FUNCTION_BLOCK FB_Schrittbetrieb
VAR_INPUT
	eAblaufStatus:			AblaufStatus;
	eHolStatus:				AblaufStatus;
	eBereitstellStatus:		AblaufStatus;
	bAblaufAktiv:			BOOL;				//Info ob ein Teil bearbetet, geholt oder bereitgestellt werden muss
	
	bAktorPosNIO:			BOOL;				//True wenn ein aktor im handbetrieb verfahren wurde
	
	stStationInfo:			REFERENCE TO ST_Station;
	bRstInPos:				BOOL;
END_VAR
VAR_OUTPUT
	bInQueue:				BOOL;				//Es wurde rueckwaerts in die Queue gefahren und die vorherige Position wurde nicht wieder erreicht
	bAblaufFreigabe:		BOOL;				//Die Aktoren im normalen Ablauf dürfen fahren (Handoverride true) (nur bis Statuswechsel true)
	bSendFalschePosError:	BOOL;				//Aktoren sollen falsche Pos senden
END_VAR
VAR
	aSchrittQueue:			ARRAY[0..Parameter.cGroesseSchrittQueue] OF ST_SchrittQueue;
	nIndex:					INT;
	i:						INT;
	
	nAktPosition:			INT;				//Aktuelle Position in Queue
	nSollAktPos:			INT;				//Welche position andgefahren werden soll (wechselt schon wenn bewegung ausgefuehrt aber Sensoren nicht angeben)
	
	
	ePrevAblaufStatus:		AblaufStatus;
	ePrevHolStatus:			AblaufStatus;	
	ePrevBereitstellStatus:	AblaufStatus;
	
	bBtnSchrittVor:			BOOL;
	bBtnSchrittZurueck:		BOOL;
	
	bSchrittVor:			BOOL;
	bSchrittZurueck:		BOOL;
	bVorBisEnde:			BOOL;
	
	fbSendErrorTrig:		R_TRIG;
END_VAR

//********************************************************************************
//Statuswechsel erkennen
IF			ePrevAblaufStatus <> eAblaufStatus
	OR		ePrevHolStatus <> eHolStatus
	OR		ePrevBereitstellStatus <> eBereitstellStatus THEN
	
	IF			nIndex > 0 THEN
		aSchrittQueue[nIndex-1].bStatuswechsel := TRUE;
	END_IF
	
	bAblaufFreigabe := FALSE;
	
	ePrevAblaufStatus		:= eAblaufStatus;
	ePrevHolStatus			:= eHolStatus;
	ePrevBereitstellStatus	:= eBereitstellStatus;
END_IF

//********************************************************************************
//Handheld
IF			MAIN.fbHandheld.nGewaehlteStation = stStationInfo.nStationsNr THEN
	
	IF			MAIN.bE_Handbetrieb THEN
		
		IF			MAIN.fbHandheld.fbVorTrig.Q THEN
			bBtnSchrittVor := TRUE;
		ELSIF		MAIN.fbHandheld.fbZurueckTrig.Q THEN
			bBtnSchrittZurueck := TRUE;
		END_IF
		
	END_IF
END_IF

//********************************************************************************
//Zurueck zu Start wenn Anlage weiterlaeuft
IF			MAIN.bProduzieren
	AND NOT MAIN.bE_Handbetrieb
	AND		bInQueue
	AND NOT bSchrittZurueck
	AND NOT bSchrittVor THEN
	bVorBisEnde := TRUE;
	bBtnSchrittVor := TRUE;
ELSIF		MAIN.bE_Handbetrieb
	OR	NOT bInQueue THEN
	bVorBisEnde := FALSE;
END_IF

//********************************************************************************
//Aktoren fehler senden lassen wenn pos NIO 
fbSendErrorTrig(CLK := 			bAktorPosNIO 
						AND		(bBtnSchrittVor 
						OR 		bBtnSchrittZurueck),
				Q => bSendFalschePosError);

//********************************************************************************
//Schrittausloesung
IF 		NOT MAIN.bE_Handbetrieb THEN		//Zurück geht nur im Handbetrieb (vor geht auch wenn bis zum Ende gefahren weden mus)
	bBtnSchrittZurueck := FALSE;
END_IF

IF			(MAIN.bE_Handbetrieb
	OR		bVorBisEnde)
	AND	NOT bAktorPosNIO THEN
	
	IF			bBtnSchrittVor THEN
		bBtnSchrittVor := FALSE;
		
		IF			bSchrittZurueck THEN
			bSchrittZurueck := FALSE;
			nAktPosition := nSollAktPos;
		END_IF
	
		bSchrittVor := TRUE;			//Kann nur gesetzt werden wenn bSchrittZueuck nicht gesetzt ist
	END_IF
	
	IF			bBtnSchrittZurueck THEN
		bBtnSchrittZurueck := FALSE;
		
		//Wenn ein Schritt im Ablauf nicht fertig wird kann trozdem zurueck gefahren werden
		IF			bAblaufFreigabe THEN
			bAblaufFreigabe := FALSE;
		END_IF
		
		IF			bSchrittVor THEN
			bSchrittVor := FALSE;
			nAktPosition := nSollAktPos;
		END_IF
		
		bSchrittZurueck := TRUE;			//Kann nur gesetzt werden wenn bSchrittZueuck nicht gesetzt ist
	END_IF
ELSE
	bBtnSchrittVor := FALSE;
	bBtnSchrittZurueck := FALSE;
	bAblaufFreigabe := FALSE;
END_IF

//********************************************************************************
//Aktor Pos NIO reset damit die aktoren erneut setzen koennen im naechsten zuecklus
bAktorPosNIO := FALSE;

//********************************************************************************
//Schrittauslösung Ausführen
IF			bSchrittVor THEN
	bSchrittVor := NOT schrittVor();
END_IF

IF			bSchrittZurueck THEN
	bSchrittZurueck := NOT schrittZurueck();
END_IF

METHOD addToQueue
VAR_INPUT
	stEintrag:			ST_SchrittQueue;
END_VAR
VAR
	i:					INT;
END_VAR
//Bewegungen nicht aufnehmen wenn in der Queue verfahren wird
IF			bInQueue
	OR		bSchrittVor
	OR		bSchrittZurueck THEN
	RETURN;
END_IF


IF			(nIndex > Parameter.cGroesseSchrittQueue) THEN
	nIndex := Parameter.cGroesseSchrittQueue;
	
	//Alle Eintraege schieben, aelteste faellt raus
	FOR i:=1 TO Parameter.cGroesseSchrittQueue DO
		aSchrittQueue[i-1] := aSchrittQueue[i];
	END_FOR
END_IF

//In Queue aufnehmen und Message zurueckgeben
aSchrittQueue[nIndex] := stEintrag;
nAktPosition := nIndex;
nIndex := nIndex+1;
END_METHOD

METHOD reset
VAR_INPUT
END_VAR
VAR
	i:						INT;
	stTempLeer:				ST_SchrittQueue;
END_VAR
//Alle Eintraege schieben, aelteste faellt raus
FOR i:=0 TO Parameter.cGroesseSchrittQueue DO
	aSchrittQueue[i] := stTempLeer;
END_FOR
nIndex 			:= 0;
nAktPosition 	:= 0;
bInQueue 		:= FALSE;
bSchrittVor 	:= FALSE;
bSchrittZurueck := FALSE;
bAblaufFreigabe := FALSE;
END_METHOD

METHOD PRIVATE schrittVor : BOOL
VAR_INPUT
END_VAR
VAR
	i:						INT;
	nIndexbStatuswechsel:	INT;
	bPosErreicht: 			BOOL;
END_VAR
IF		NOT bRstInPos THEN
	RETURN;
END_IF

//return wenn Ende erreicht
IF			nAktPosition >= (nIndex-1) THEN
	bAblaufFreigabe := bAblaufAktiv;
	bInQueue := FALSE;
	schrittVor := TRUE;
	RETURN;
END_IF

//********************************************************************************
FOR i:= nAktPosition+1 TO nIndex-1 DO	
	nIndexbStatuswechsel := i;
	nSollAktPos := i;					//Ist immer aktuell wenn for verlassen wird
	
	IF 			aSchrittQueue[i].bGesetzt THEN			
		//*****************************************************************
		IF			__ISVALIDREF(aSchrittQueue[i].fbAktor) THEN
			aSchrittQueue[i].fbAktor.bHandOverride := TRUE;
			aSchrittQueue[i].bInPos := aSchrittQueue[i].fbAktor.arbeitsPos();
			aSchrittQueue[i].fbAktor.bHandOverride := FALSE;
		ELSIF		__ISVALIDREF(aSchrittQueue[i].fbOutput) THEN
			aSchrittQueue[i].fbOutput.bHandOverride := TRUE;
			aSchrittQueue[i].bInPos := aSchrittQueue[i].fbOutput.set();
			aSchrittQueue[i].fbOutput.bHandOverride := FALSE;
		ELSE
			//Fehler!!!
			i := i-1;
			EXIT;
		END_IF
		//*****************************************************************
	ELSE
		//*****************************************************************
		IF			__ISVALIDREF(aSchrittQueue[i].fbAktor) THEN
			aSchrittQueue[i].fbAktor.bHandOverride := TRUE;
			aSchrittQueue[i].bInPos := aSchrittQueue[i].fbAktor.ruhePos();
			aSchrittQueue[i].fbAktor.bHandOverride := FALSE;
		ELSIF		__ISVALIDREF(aSchrittQueue[i].fbOutput) THEN
			aSchrittQueue[i].fbOutput.bHandOverride := TRUE;
			aSchrittQueue[i].bInPos := aSchrittQueue[i].fbOutput.reset();
			aSchrittQueue[i].fbOutput.bHandOverride := FALSE;
		ELSE
			//Fehler!!!
			i := i-1;
			EXIT;
		END_IF
		//*****************************************************************
	END_IF
	
	IF		aSchrittQueue[i].bStatuswechsel THEN
		EXIT;
	END_IF
END_FOR

//********************************************************************************
bPosErreicht := TRUE;
FOR i:= nAktPosition+1 TO nIndexbStatuswechsel DO
	IF		NOT	aSchrittQueue[i].bInPos THEN
		bPosErreicht := FALSE;
	END_IF
END_FOR

//Alle inPos bei jedem Aufruf zuruecksetzten
FOR i:= nAktPosition+1 TO nIndexbStatuswechsel DO
	aSchrittQueue[i].bInPos := FALSE;
END_FOR

IF			bPosErreicht THEN
	nAktPosition := nIndexbStatuswechsel;
	IF			nAktPosition = (nIndex-1) THEN
		bInQueue := FALSE;
	END_IF	
	schrittVor := TRUE;	
END_IF
END_METHOD

METHOD PRIVATE schrittZurueck : BOOL
VAR_INPUT
END_VAR
VAR
	i:						INT;
	nIndexbStatuswechsel:	INT;
	bPosErreicht: 			BOOL;
	
	nPosVorher:				INT;
END_VAR
IF		NOT bRstInPos THEN
	RETURN;
END_IF

IF			nAktPosition >= 0 THEN
	bInQueue := TRUE;
ELSE									//Wenn noch kein Schritt aufgezeichnet wurde -> return True
	schrittZurueck := TRUE;
	RETURN;
END_IF

//********************************************************************************
FOR i:= nAktPosition TO 0 BY -1 DO
	nIndexbStatuswechsel := i;
	nSollAktPos := i;					//Ist immer aktuell wenn for verlassen wird

	IF		NOT aSchrittQueue[i].bStatuswechsel
		OR		i = nAktPosition THEN
			
		IF 			aSchrittQueue[i].bGesetzt THEN			
			//*****************************************************************
			IF			__ISVALIDREF(aSchrittQueue[i].fbAktor) THEN
				aSchrittQueue[i].fbAktor.bHandOverride := TRUE;
				aSchrittQueue[i].bInPos := aSchrittQueue[i].fbAktor.ruhePos();
				aSchrittQueue[i].fbAktor.bHandOverride := FALSE;
			ELSIF		__ISVALIDREF(aSchrittQueue[i].fbOutput) THEN
				aSchrittQueue[i].fbOutput.bHandOverride := TRUE;
				aSchrittQueue[i].bInPos := aSchrittQueue[i].fbOutput.reset();
				aSchrittQueue[i].fbOutput.bHandOverride := FALSE;
			ELSE
				//Fehler!!!
				EXIT;
			END_IF
			//*****************************************************************
		ELSE
			//*****************************************************************
			IF			__ISVALIDREF(aSchrittQueue[i].fbAktor) THEN
				aSchrittQueue[i].fbAktor.bHandOverride := TRUE;
				aSchrittQueue[i].bInPos := aSchrittQueue[i].fbAktor.arbeitsPos();
				aSchrittQueue[i].fbAktor.bHandOverride := FALSE;
			ELSIF		__ISVALIDREF(aSchrittQueue[i].fbOutput) THEN
				aSchrittQueue[i].fbOutput.bHandOverride := TRUE;
				aSchrittQueue[i].bInPos := aSchrittQueue[i].fbOutput.set();
				aSchrittQueue[i].fbOutput.bHandOverride := FALSE;
			ELSE
				//Fehler!!!
				EXIT;
			END_IF
			//*****************************************************************
		END_IF
		
		//Wenn i=0 ist und der Schritt in Queue[0] ausgeführt wurde muss index -1 sein damit Queue[0] beim vorwärts fahren wieder ausgeführt wird
		IF			i = 0 THEN
			nIndexbStatuswechsel := -1;
			nSollAktPos := -1;
		END_IF
		
	ELSIF		aSchrittQueue[i].bStatuswechsel
		AND		i <> nAktPosition THEN
		EXIT;
	END_IF
END_FOR

//********************************************************************************
//Abfrage alle in Pos
bPosErreicht := TRUE;
FOR i:= nAktPosition TO nIndexbStatuswechsel+1 BY -1 DO
	IF		NOT	aSchrittQueue[i].bInPos THEN
		bPosErreicht := FALSE;
	END_IF
END_FOR

//Alle inPos bei jedem Aufruf zuruecksetzten
FOR i:= nAktPosition TO nIndexbStatuswechsel+1 BY -1 DO
	aSchrittQueue[i].bInPos := FALSE;
END_FOR

IF			bPosErreicht THEN
	nAktPosition := nIndexbStatuswechsel;
	schrittZurueck := TRUE;
END_IF
END_METHOD

METHOD vor
VAR_INPUT
END_VAR
bBtnSchrittVor := TRUE;
END_METHOD

METHOD zurueck
VAR_INPUT
END_VAR
bBtnSchrittZurueck := TRUE;
END_METHOD

END_FUNCTION_BLOCK

(* stored: Version 1.1.0.1, ProductVersion 3.1.4024.12
   POU FB_Schrittbetrieb: Id {49267e6f-7334-4a2c-8702-a1c7cf9626d3}, SpecialFunc None
   Method addToQueue: Id {76ed82ee-18f3-436d-8f4a-493059dd1613}
   Method reset: Id {f62ec5d3-ef61-4923-8692-a04401c32f54}
   Method schrittVor: Id {a1184994-5b83-4a87-9d10-6132d4050c03}
   Method schrittZurueck: Id {2f0e8325-71fc-42d2-9385-f93f92b020e7}
   Method vor: Id {af8b32c6-933a-4093-ae38-5aed81f2accf}
   Method zurueck: Id {4bf4315e-4bc7-4ac8-b37a-be7a9ae2530c} *)
